FUNCTION_BLOCK FB_MotionAxisCommon IMPLEMENTS I_MotionAxisCommon
VAR_INPUT
END_VAR
VAR_OUTPUT
END_VAR
VAR

    {attribute 'no_copy'}
    AxisRef : REFERENCE TO AXIS_REF;
    stMotionDriveReference : REFERENCE TO ST_MotionDrive;
    stMotionEpicsInterfaceReference : REFERENCE TO ST_MotionEpicsInterface;

    mcReadParams: MC_ReadParameterSet;
    // MC_ReadParameterSet Output
    stAxisParameters: ST_AxisParameterSet;
    stAxisParameterSetExposed : ST_AxisParameterSetExposed;
    bNcParamsReadDone   : BOOL;
    bError				: BOOL;
    nErrorCode			: UDINT;
    nEncoderCount 		: UDINT;
END_VAR

THIS^.NCParams(TRUE, tRefreshDelay:=T#1S);
THIS^.CalibrateRawEncValue();

{warning 'Add property implementation'}
PROPERTY AxisParameterSetExposed : ST_AxisParameterSetExposed
GET
AxisParameterSetExposed := stAxisParameterSetExposed;
END_GET
SET
stAxisParameterSetExposed := AxisParameterSetExposed;
END_SET
END_PROPERTY

METHOD CalibrateRawEncValue
// IF init failed to get a valid reference then dont proceed here.
IF NOT __ISVALIDREF(stMotionDriveReference) OR NOT __ISVALIDREF(stMotionEpicsInterfaceReference) THEN
    RETURN;
END_IF

IF stMotionDriveReference.nRawEncoderULINT <> 0 THEN
    IF stMotionDriveReference.nRawEncoderULINT < 4294967296 THEN
        stMotionEpicsInterfaceReference.nEncoderCount := ULINT_TO_UDINT(stMotionDriveReference.nRawEncoderULINT);
    ELSE
        stMotionEpicsInterfaceReference.nEncoderCount := ULINT_TO_UDINT(18446744073709551615 - stMotionDriveReference.nRawEncoderULINT);
    END_IF
ELSIF stMotionDriveReference.nRawEncoderUINT <> 0 THEN
    stMotionEpicsInterfaceReference.nEncoderCount := UINT_TO_UDINT(stMotionDriveReference.nRawEncoderUINT);
ELSIF stMotionDriveReference.nRawEncoderINT <> 0 THEN
    stMotionEpicsInterfaceReference.nEncoderCount := INT_TO_UDINT(stMotionDriveReference.nRawEncoderINT);
ELSIF stMotionDriveReference.nRawEncoderDINT <> 0 THEN
    stMotionEpicsInterfaceReference.nEncoderCount := DINT_TO_UDINT(stMotionDriveReference.nRawEncoderDINT);
ELSE
    stMotionEpicsInterfaceReference.nEncoderCount := 0;
END_IF
END_METHOD

{warning 'Add property implementation'}
PROPERTY EncoderCount : UDINT
GET
EncoderCount := nEncoderCount;
END_GET
SET
nEncoderCount := EncoderCount;
END_SET
END_PROPERTY

PROPERTY Error : BOOL
GET
Error := bError;
END_GET
SET
bError := Error;
END_SET
END_PROPERTY

PROPERTY ErrorCode : UDINT
GET
ErrorCode := nErrorCode;
END_GET
SET
nErrorCode := ErrorCode;
END_SET
END_PROPERTY

//FB_Init is always available implicitly and it is used primarily for initialization.
//The return value is not evaluated. For a specific influence, you can also declare the
//methods explicitly and provide additional code there with the standard initialization
//code. You can evaluate the return value.
METHOD FB_Init: BOOL
VAR_INPUT
    bInitRetains: BOOL; // TRUE: the retain variables are initialized (reset warm / reset cold)
    bInCopyCode: BOOL;  // TRUE: the instance will be copied to the copy code afterward (online change)
    AxisReference : REFERENCE TO AXIS_REF;
END_VAR
AxisRef REF= AxisReference;
END_METHOD

METHOD GetDriveAndEpicsItfRefs
VAR_INPUT
    stMotionDriveRef : REFERENCE TO ST_MotionDrive;
    stMotionEpicsInterfaceRef : REFERENCE TO ST_MotionEpicsInterface;
END_VAR
    stMotionDriveReference REF= stMotionDriveRef;
    stMotionEpicsInterfaceReference REF= stMotionEpicsInterfaceRef;
END_METHOD

METHOD NCParams : BOOL;
VAR_INPUT
    bEnable: BOOL;
    tRefreshDelay: TIME;
END_VAR

VAR_INST
    timer: TON;
    bExecute: BOOL := TRUE;
    nLatchErrId: UDINT;
END_VAR
timer(
    IN:=bEnable AND NOT bExecute,
    PT:=tRefreshDelay);
bExecute S= timer.Q;
mcReadParams(
    Parameter:=THIS^.stAxisParameters,
    Axis:= AxisRef,
    Execute:=bEnable AND bExecute );

IF mcReadParams.Error THEN
    Error := TRUE;
    ErrorCode := mcReadParams.ErrorID;
    // Log this error
END_IF

(* IF mcReadParams.ErrorID <> 0 THEN
    nLatchErrId := 0;
END_IF *)

// Copy axis parameters that we want to expose to the EPICS layer.
THIS^.stAxisParameterSetExposed.bCtrlEnablePosDiffControl     := THIS^.stAxisParameters.bCtrlEnablePosDiffControl;
THIS^.stAxisParameterSetExposed.bEncEnableSoftEndMaxControl   := THIS^.stAxisParameters.bEncEnableSoftEndMaxControl;
THIS^.stAxisParameterSetExposed.bEncEnableSoftEndMinControl   := THIS^.stAxisParameters.bEncEnableSoftEndMinControl;
THIS^.stAxisParameterSetExposed.fAccelerationMax              := THIS^.stAxisParameters.fAccelerationMax;
THIS^.stAxisParameterSetExposed.fCtrlPosDiffMax               := THIS^.stAxisParameters.fCtrlPosDiffMax;
THIS^.stAxisParameterSetExposed.fCtrlPosDiffMaxTime           := THIS^.stAxisParameters.fCtrlPosDiffMaxTime;
THIS^.stAxisParameterSetExposed.fDecelerationMax              := THIS^.stAxisParameters.fDecelerationMax;
THIS^.stAxisParameterSetExposed.fEncSoftEndMax                := THIS^.stAxisParameters.fEncSoftEndMax;
THIS^.stAxisParameterSetExposed.fEncSoftEndMin                := THIS^.stAxisParameters.fEncSoftEndMin;
THIS^.stAxisParameterSetExposed.fVeloMaximum                  := THIS^.stAxisParameters.fVeloMaximum;
THIS^.stAxisParameterSetExposed.fEncOffset               	  := THIS^.stAxisParameters.fEncOffset;
THIS^.stAxisParameterSetExposed.fEncScaleFactorInternal       := THIS^.stAxisParameters.fEncScaleFactorInternal;

bExecute R= mcReadParams.Done OR mcReadParams.Error;
NCParamsReadDone S= mcReadParams.Done;
END_METHOD

PROPERTY NCParamsReadDone : BOOL
GET
NCParamsReadDone := bNCParamsReadDone;
END_GET
SET
bNCParamsReadDone := NCParamsReadDone;
END_SET
END_PROPERTY

END_FUNCTION_BLOCK

(* stored: Version 1.1.0.1
   POU FB_MotionAxisCommon: Id {b2f4c148-bcde-4ca5-a7a9-abd4413ce8ab}, SpecialFunc None
   Property AxisParameterSetExposed: Id {bd38f88c-c219-4363-856f-6d4d63c13ec4}
   Get Get: Id {50330633-1a97-458e-b8ef-ffa028d8a61b}
   Set Set: Id {6b74fee6-0826-4088-8509-987679c32e97}
   Method CalibrateRawEncValue: Id {1731f1b4-fc8d-48cd-81d7-d75b2a571773}
   Property EncoderCount: Id {5225d004-dac1-4dfa-90f6-2aa283ea59c1}
   Get Get: Id {4699599a-607a-4379-8415-7f67e45880a3}
   Set Set: Id {5916a47b-3bdc-477b-b2e2-fa22d0699a1c}
   Property Error: Id {2819c2f0-b6fd-42b1-b42d-175038209c48}
   Get Get: Id {c757a456-f781-4926-9229-39a5572ee16c}
   Set Set: Id {ccc50871-05d6-40ce-aca3-048fcd2bfa2b}
   Property ErrorCode: Id {b7569608-1ea8-4914-a3b4-543b15f7c860}
   Get Get: Id {37935438-07d0-4e35-a5a0-50e5e1f3d03b}
   Set Set: Id {53062068-e81d-4dce-b763-5cd409ed4079}
   Method FB_Init: Id {8bc50fb9-2f4e-4094-860c-18b3654dc16c}
   Method GetDriveAndEpicsItfRefs: Id {521243a9-080c-4717-80a3-4aef48e01826}
   Method NCParams: Id {dd5f801a-4004-4e64-a8a8-d3052d398ddb}
   Property NCParamsReadDone: Id {fc8144c2-ca29-4700-853c-a4a1e0fc319a}
   Get Get: Id {bf6c53f4-cc0b-4a81-96a0-d612250516fd}
   Set Set: Id {05cf4a9b-1c44-4464-9615-25d3dfbdef0f} *)
